// TIA Portal V20 export
FUNCTION_BLOCK "FB_AnalogInputThreshold"   // FB221, SCL
{ S7_Optimized_Access := 'TRUE' }
// stored: AutoNumber false, MemoryReserve 100, SetENOAutomatically false
   VAR_INPUT
      iActualValue : Real;
      iStartDelay : Bool;
      iDataPLC { ExternalAccessible := 'False'; ExternalVisible := 'False'; ExternalWritable := 'False'} : "AnalogInDataPLC_DT";
      iDataHMI { ExternalAccessible := 'False'; ExternalVisible := 'False'; ExternalWritable := 'False'} : "AnalogInDataHMI_DT";
   END_VAR
   VAR_OUTPUT
      oDataAction { ExternalAccessible := 'False'; ExternalVisible := 'False'; ExternalWritable := 'False'} : "AnalogInAction_DT";
   END_VAR
   VAR_IN_OUT
      ioAlarmMin : Bool;
      ioWarningMin : Bool;
      ioWarningMax : Bool;
      ioAlarmMax : Bool;
   END_VAR
   VAR
      sStartTimer : TON_TIME;
      sTONAlarmMin : TON_TIME;
      sTONWarningMin : TON_TIME;
      sTONWarningMax : TON_TIME;
      sTONAlarmMax : TON_TIME;
      sMemoAlarmMin { S7_SetPoint := 'True'} : Bool;
      sMemoWarningMin { S7_SetPoint := 'True'} : Bool;
      sMemoWarningMax { S7_SetPoint := 'True'} : Bool;
      sMemoAlarmMax { S7_SetPoint := 'True'} : Bool;
   END_VAR
BEGIN
   REGION Description header 
       //==================================================================================
       // POSALUX Swiss SA / (C) Copyright 2024
       //----------------------------------------------------------------------------------
       // Title: Analog input management 
       // Comment/Function: This function manages alarms and warnings based on a  
       //                   current value compared to predefined target. After an
       //                   initial delay, it activates specific alarms OR warnings if the
       //                   value exceeds thresholds, and can also trigger machine
       //                   shutdown or signal a defective part according TO conditions
       //                   configured on the HMI.
       // Author: Gowsigan SRITHARAN
       // Engineering: TIA Portal v17
       //----------------------------------------------------------------------------------
       // Change log table:
       // Version  | Date     | Expert in charge | Changes applied
       // ---------|----------|------------------|------------------------------------
       // 00.00.01 | 20241121 | GSR              | First released version
       // 00.00.02 | 20250911 | WFA              | Work with target
       // ==================================================================================
   END_REGION

   REGION Start Timer
       #sStartTimer(IN := #iStartDelay,
                    PT := #iDataHMI.StartTime);
       #sTONAlarmMin(IN := #sMemoAlarmMin,
                     PT := #iDataPLC.DelayAlarmMin);
       #sTONWarningMin(IN := #sMemoWarningMin,
                       PT := #iDataPLC.DelayWarningMin);
       #sTONAlarmMax(IN := #sMemoAlarmMax,
                     PT := #iDataPLC.DelayAlarmMax);
       #sTONWarningMax(IN := #sMemoWarningMax,
                       PT := #iDataPLC.DelayWarningMax);
   END_REGION

   REGION Detect alarm/warning
       IF #sStartTimer.Q THEN
           #sMemoWarningMin := #iDataHMI.TargetValue + #iDataHMI.ThresholdWarningMin >= #iActualValue AND #iDataPLC.EnableWarningMin AND NOT #sMemoAlarmMin;

           #sMemoWarningMax := #iDataHMI.TargetValue + #iDataHMI.ThresholdWarningMax <= #iActualValue AND #iDataPLC.EnableWarningMax AND NOT #sMemoAlarmMax;

           #sMemoAlarmMin := #iDataHMI.TargetValue + #iDataHMI.ThresholdAlarmMin >= #iActualValue AND #iDataPLC.EnableAlarmMin;

           #sMemoAlarmMax := #iDataHMI.TargetValue + #iDataHMI.ThresholdAlarmMax <= #iActualValue AND #iDataPLC.EnableAlarmMax;
       ELSE
           #sMemoWarningMin := FALSE;
           #sMemoWarningMax := FALSE;
           #sMemoAlarmMin   := FALSE;
           #sMemoAlarmMax   := FALSE;
       END_IF;

   END_REGION

   REGION Set alarm/warning
       // Alarme Min
       IF #sTONAlarmMin.Q THEN
           #ioAlarmMin := TRUE;
           #ioWarningMin := FALSE;
           #oDataAction.BadPartOnFixture := #iDataPLC.BadPartOnFixture; // Set bad part if alarm
           #oDataAction.ID_Measure := #iDataHMI.ID_Measure;
       ELSE
           #oDataAction.BadPartOnFixture := FALSE;
           #oDataAction.ID_Measure := 0;
       END_IF;

       // Warning Min
       IF #sTONWarningMin.Q THEN
           #ioWarningMin := TRUE;
       END_IF;

       // Alarm Max
       IF #sTONAlarmMax.Q THEN
           #ioAlarmMax := TRUE;
           #ioWarningMax := FALSE;
           #oDataAction.BadPartOnFixture := #iDataPLC.BadPartOnFixture; // Set bad part if alarm
           #oDataAction.ID_Measure := #iDataHMI.ID_Measure;
       ELSE
           #oDataAction.BadPartOnFixture := FALSE;
           #oDataAction.ID_Measure := 0;
       END_IF;

       // Warning Max
       IF #sTONWarningMax.Q THEN
           #ioWarningMax := TRUE;
       END_IF;
   END_REGION
END_FUNCTION_BLOCK
